FUNCTION_BLOCK INFO
VAR_INPUT
END_VAR
VAR_OUTPUT
END_VAR
VAR
END_VAR

Couter_R_TRIG(
CLK:= , 
Q=> );

END_FUNCTION_BLOCK

(* stored: Version 1.1.0.1, ProductVersion 3.1.4024.12
   POU INFO: Id {7395f367-245f-4505-b18a-cedd56194bd6}, SpecialFunc None *)
